# EPICS autosave request: iocBoot/gmca_23b_ioc2/dbSave/drv1.req
%
% BURT Request File
%
% AXIS
%

% RO $(DRV1):ActPos
$(DRV1):ActPos.EGU
$(DRV1):ActPos.DESC

$(DRV1):RqsPos
$(DRV1):RqsPos.EGU
$(DRV1):RqsPos.DESC
$(DRV1):RqsPos.HOPR
$(DRV1):RqsPos.LOPR
$(DRV1):RqsPos.DRVH
$(DRV1):RqsPos.DRVL

$(DRV1):RqsBkl
$(DRV1):RqsBkl.EGU
$(DRV1):RqsBkl.DESC

$(DRV1):RqsPosInc
$(DRV1):MemPos

$(DRV1):Offset
$(DRV1):Scale
